FUNCTION_BLOCK L3_OrderTable (* Service Interface Function Block Type *)
  (* Standard: 61499-2; Description: This SIFB holds a table where are stacked all manufacturing orders. Table is updated every time that an individual part is completed. *)
  (* Version 0.0, 2014-09-29, EQUEROL, UJI *)
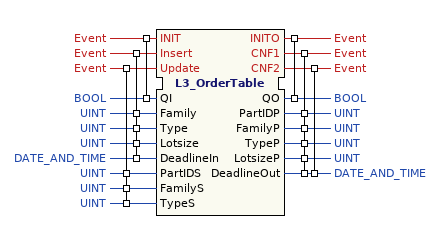
  EVENT_INPUT
    INIT WITH QI; (* Service Initialization *)
    Insert WITH Family, Type, Lotsize, DeadlineIn; (* Insert a new order into the table *)
    Update WITH PartIDS, FamilyS, TypeS; (* Update the table with manufacturing results *)
  END_EVENT
  EVENT_OUTPUT
    INITO WITH QO; (* Initialization Confirm *)
    CNF1 WITH PartIDP, FamilyP, TypeP, LotsizeP, DeadlineOut; (* Confirmation of insertion *)
    CNF2 WITH DeadlineOut; (* confirmation of update *)
  END_EVENT
  VAR_INPUT
    QI : BOOL; (* Event Input Qualifier *)
    Family : UINT; (* Part's family *)
    Type : UINT; (* Part's type *)
    Lotsize : UINT; (* Number of parts to be manufactured *)
    DeadlineIn : DATE_AND_TIME; (* Deadline of the lot to be inserted *)
    PartIDS : UINT; (* Part Identifier *)
    FamilyS : UINT; (* Part's family *)
    TypeS : UINT; (* Part's type *)
  END_VAR
  VAR_OUTPUT
    QO : BOOL; (* Event Output Qualifier *)
    PartIDP : UINT; (* Part identifier *)
    FamilyP : UINT; (* Part's family *)
    TypeP : UINT; (* Part's type *)
    LotsizeP : UINT; (* lot size *)
    DeadlineOut : DATE_AND_TIME; (* Updated deadline *)
  END_VAR
  SERVICE APPLICATION/RESOURCE (* Service Interface Function Block Type *)
    SEQUENCE normal_establishment
      APPLICATION.INIT+(PARAMS) -> APPLICATION.INITO+(PARAMS);
    END_SEQUENCE
    SEQUENCE unsuccessful_establishment
      APPLICATION.INIT+(PARAMS) -> APPLICATION.INITO-(STATUS);
    END_SEQUENCE
    SEQUENCE insertion_confirm
      APPLICATION.Insert(SD) -> APPLICATION.CNF1(RD);
    END_SEQUENCE
    SEQUENCE application_initiated_termination
      APPLICATION.INIT-() -> APPLICATION.INITO-(STATUS);
    END_SEQUENCE
    SEQUENCE resource_initiated_termination
      -> APPLICATION.INITO-(STATUS);
    END_SEQUENCE
    SEQUENCE update_confirm
      APPLICATION.Update() -> APPLICATION.CNF2();
    END_SEQUENCE
  END_SERVICE
END_FUNCTION_BLOCK
